// TIA Portal V20 export
DATA_BLOCK "InstCallAlarmCounter"   // DB25
// stored: InstanceOfName CallAlarmCounter, InstanceOfType FB
"CallAlarmCounter"
   // VAR
   //    statPulse { ExternalAccessible := 'False'; ExternalVisible := 'False'; ExternalWritable := 'False'} : Array[0..99] of Bool;
   // END_VAR
BEGIN
END_DATA_BLOCK
